{attribute 'GeneratedUsingTerminal: '}
{attribute addProperty BoxType ""}
{attribute addProperty Id ""}
{attribute addProperty CRC "0"}
{attribute addProperty Size "0"}
TYPE EtcSlaveTerminalBase :
STRUCT
END_STRUCT
END_TYPE

(* stored: Version 1.2.0.0, ProductVersion 3.1.4024.9
   DUT EtcSlaveTerminalBase: Id {b9332a0a-0c01-4473-a306-60ee30e088fd} *)
